// TIA Portal V15.1 export
// export: Created 2024-05-17T05:38:20.1338175Z, ExportSetting WithDefaults, DisplayName Totally Integrated Automation Portal, DisplayVersion V15.1 Update 5, DisplayName TIA Portal Openness, DisplayVersion V15.1 Update 5, DisplayName SINAMICS Startdrive Advanced, DisplayVersion V15.1, DisplayName G130, G150, S120, S150, SINAMICS MV, S210, DisplayVersion V15.1, DisplayName G110M, G120, G120C, G120D, G120P, DisplayVersion V15.1, DisplayName STEP 7 Professional, DisplayVersion V15.1 Update 5, DisplayName STEP 7 Safety, DisplayVersion V15.1, DisplayName WinCC Professional, DisplayVersion V15.1 Update 5, DisplayName SIMATIC Visualization Architect, DisplayVersion V15.1
DATA_BLOCK "_209220ZM01Config"   // DB352
{ S7_Optimized_Access := 'FALSE' }
AUTHOR : VCC
VERSION : 0.1
// stored: AutoNumber false, DBAccessibleFromOPCUA true, IsOnlyStoredInLoadMemory false, IsWriteProtectedInAS false
   VAR
      Andon { ExternalAccessible := 'False'; ExternalVisible := 'False'; ExternalWritable := 'False'} : "AndonConfigVCG";   // Config
      "220CS22ProdSpeed" { ExternalAccessible := 'False'; ExternalVisible := 'False'; ExternalWritable := 'False'} : "ProdSpeedConfig";   // Config
      "220CS22ProdStartStop" { ExternalAccessible := 'False'; ExternalVisible := 'False'; ExternalWritable := 'False'} : "ProdStartStopConfig";   // Config
      "220CS22LineFeed" { ExternalAccessible := 'False'; ExternalVisible := 'False'; ExternalWritable := 'False'} : "LineFeedConfig";   // Config
      "220CS22ShiftRegLine" { ExternalAccessible := 'False'; ExternalVisible := 'False'; ExternalWritable := 'False'} : "ShiftRegLineConfig";   // Config
      "220CHB21" { ExternalAccessible := 'False'; ExternalVisible := 'False'; ExternalWritable := 'False'} : "MovUnit2Pos2S-MoviFitFCPNConfig";   // Config
      "220CR21" { ExternalAccessible := 'False'; ExternalVisible := 'False'; ExternalWritable := 'False'} : "RollerConvMDXPNConfig";   // Config
      "220CS22" { ExternalAccessible := 'False'; ExternalVisible := 'False'; ExternalWritable := 'False'} : "LineConvBrake-MDXPNConfig";   // Config
      "220CR23" { ExternalAccessible := 'False'; ExternalVisible := 'False'; ExternalWritable := 'False'} : "RollerConvMDXPNConfig";   // Config
      "220ASH01" { ExternalAccessible := 'False'; ExternalVisible := 'False'; ExternalWritable := 'False'} : "HandHeldHBA-Config";   // Config
   END_VAR
BEGIN
END_DATA_BLOCK
